# B&R Automation Studio project PLC_base3
Automation Studio 4.8.2.72

## Logical view

### Global.var - Global variables
```iecst
VAR
	data1 : STRING[1000];
	data2 : STRING[1000];
	activeData : USINT;
	readyForData : BOOL;
	receivedData : BOOL;
	readyToConvert : BOOL;
	instSize : DINT;
	instructionsArray : ARRAY[0..999] OF STRING[25];
	xArray : ARRAY[0..999] OF INT;
	yArray : ARRAY[0..999] OF INT;
	zArray : ARRAY[0..999] OF INT;
END_VAR
```

### Program Logical/Program (IEC)

#### Main.st - Init, cyclic, exit code
```iecst
PROGRAM _INIT
	ROBOSTATE := READY;

	counter := 0;
	delim1 := ' ';
	delim2 := ',';

	xEnable := FALSE;
	yEnable := FALSE;
	zEnable := FALSE;

	count := 0;
	xCounter := 0;
	yCounter := 0;
	zCounter := 0;
	xCalib := 0; //17680
	yCalib := 0; //13364
	zCalib := 0;
	yPrev := 0;
	xNext := FALSE;
	yNext := FALSE;
	zNext := FALSE;
	xDirection := FALSE;
	yDirection := FALSE;
	zDirection := FALSE;
	xStep := FALSE;
	yStep := FALSE;
	zStep := FALSE;
	xNegMove := FALSE;
	yNegMove := FALSE;
	zNegMove := FALSE;
	xPosMove := FALSE;
	yPosMove := FALSE;
	zPosMove := FALSE;
	hasBeenSharpened := TRUE;
	scale := 25; // steps / px
END_PROGRAM

PROGRAM _CYCLIC
	IF killswitch THEN // Killswitch to stop robot in case of emergency
		//ROBOSTATE := STOP;
	END_IF;

	CASE ROBOSTATE OF
		INIT:
			counter := 0;
			delim1 := ' ';
			delim2 := ',';

			xEnable := FALSE;
			yEnable := FALSE;
			zEnable := FALSE;

			count := 0;
			xCounter := 0;
			yCounter := 0;
			zCounter := 0;
			xCalib := 0; //17680
			yCalib := 0; //13364
			zCalib := 0;
			yPrev := 0;
			xNext := FALSE;
			yNext := FALSE;
			zNext := FALSE;
			xDirection := FALSE;
			yDirection := FALSE;
			zDirection := FALSE;
			xStep := FALSE;
			yStep := FALSE;
			zStep := FALSE;
			xNegMove := FALSE;
			yNegMove := FALSE;
			zNegMove := FALSE;
			xPosMove := FALSE;
			yPosMove := FALSE;
			zPosMove := FALSE;
			readyToConvert := FALSE;
			scale := 25;

			FOR count := 0 TO 999 DO
				instructionsArray[count] := '';
				xArray[count] := 0;
				yArray[count] := 0;
				zArray[count] := 0;
			END_FOR;

			ROBOSTATE := READY;

		READY: // Does nothing, is meant to wait until finished receiving instructions
			IF (readyToConvert = TRUE) THEN
				ROBOSTATE := CONVERT;
			END_IF

		CONVERT:
			timer(IN := NOT timer.Q, PT := T#100ms);
			IF (timer.Q = TRUE) THEN
				IF (counter < (instSize)) THEN
					// Splits element on index counter of instructionsArray[] into two seperate strings
					string1 := LEFT(instructionsArray[counter], FIND(instructionsArray[counter], delim2));
					string2 := RIGHT(instructionsArray[counter], (LEN(instructionsArray[counter]) - FIND(instructionsArray[counter], delim2)));

					// Finds numerical positions of all delimiters " " and "," in both strings
					// Isolates coordinates into individual integers
					D1 := FIND(string1, delim1);
					xString[counter] := LEFT(string1, D1 - 1);
					xArray[counter] := STRING_TO_INT(xString[counter]);
					string1 := DELETE(string1, D1, 1);

					D2 := FIND(string1, delim1);
					yString[counter] := LEFT(string1, D2 - 1);
					yArray[counter] := STRING_TO_INT(yString[counter]);
					string1 := DELETE(string1, D2, 1);

					D3 := FIND(string1, delim2);
					zString[counter] := LEFT(string1, D3 - 1);
					zArray[counter] := STRING_TO_INT(zString[counter]);

					D4 := FIND(string2, delim1);
					xString[counter + 1] := LEFT(string2, D4 - 1);
					xArray[counter + 1] := STRING_TO_INT(xString[counter + 1]);
					string2 := DELETE(string2, D1, 1);

					D5 := FIND(string2, delim1);
					yString[counter + 1] := LEFT(string2, D5 - 1);
					yArray[counter + 1] := STRING_TO_INT(yString[counter + 1]);
					string2 := DELETE(string2, D2, 1);

					D6 := FIND(string2, delim2);
					zString[counter + 1] := LEFT(string2, D6 - 1);
					zArray[counter + 1] := STRING_TO_INT(zString[counter + 1]);
					counter := counter + 2;
				ELSE
					ROBOSTATE := RESET;

					counter := 0;
				END_IF
			END_IF

		MANUAL:
			IF (killswitch <> TRUE) THEN
				IF (xStop <> TRUE OR xCounter > 0) THEN
					IF (xPosMove = TRUE) THEN
						IF (xPosMove = xNegMove) THEN
							xPosMove := FALSE;
						END_IF
						xDirection := TRUE;
						xStep := NOT xStep;
						xCounter := xCounter + 1;
					END_IF

					IF (xNegMove = TRUE) THEN
						IF (xPosMove = xNegMove) THEN
							xNegMove := FALSE;
						END_IF
						xDirection := FALSE;
						xStep := NOT xStep;
						xCounter := xCounter - 1;
					END_IF
				END_IF

				IF (yStop <> TRUE OR yCounter > 0) THEN
					IF (yPosMove = TRUE) THEN
						IF (yPosMove = yNegMove) THEN
							yPosMove := FALSE;
						END_IF
						yDirection := TRUE;
						yStep := NOT yStep;
						yCounter := yCounter + 1;
					END_IF

					IF (yNegMove = TRUE) THEN
						IF (yPosMove = yNegMove) THEN
							yNegMove := FALSE;
						END_IF
						yDirection := FALSE;
						yStep := NOT yStep;
						yCounter := yCounter - 1;
					END_IF
				END_IF

				IF (zCounter >= 0 AND zCounter <= 7500) THEN
					IF (zPosMove = TRUE) THEN
						IF (zPosMove = zNegMove) THEN
							zPosMove := FALSE;
						END_IF
						zDirection := TRUE;
						zStep := NOT zStep;
						zCounter := zCounter - 1;
					END_IF

					IF (zNegMove = TRUE) THEN
						IF (zPosMove = zNegMove) THEN
							zNegMove := FALSE;
						END_IF
						zDirection := FALSE;
						zStep := NOT zStep;
						zCounter := zCounter + 1;
					END_IF
				END_IF
			END_IF

		DRAW:
			IF (killswitch <> TRUE) OR (counter < instSize) THEN
				IF (xStop <> TRUE) THEN
					IF (xArray[counter] * scale > xCounter) THEN
						xNext := FALSE;
						xDirection := TRUE;
						xStep := NOT xStep;
						xCounter := xCounter + 1;
					ELSIF (xArray[counter] * scale < xCounter) THEN
						xNext := FALSE;
						xDirection := FALSE;
						xStep := NOT xStep;
						xCounter := xCounter - 1;
					ELSIF (xArray[counter] * scale = xCounter) THEN
						ROBOSTATE := PENCILDOWN;
					END_IF
				END_IF
			END_IF

		PENCILDOWN:
			IF (killswitch <> TRUE) THEN
				IF (bStop <> TRUE) THEN
					zDirection := TRUE;
					zStep := NOT zStep;
					zCounter := zCounter - 1;
				ELSE
					ROBOSTATE := DRAW2;
				END_IF
			END_IF

		DRAW2:
			IF (killswitch <> TRUE) THEN
				IF (xStop <> TRUE) THEN
					IF (xArray[counter + 1] * scale > xCounter) THEN
						xDirection := TRUE;
						xStep := NOT xStep;
						xCounter := xCounter + 1;
					ELSIF (xArray[counter + 1] * scale < xCounter) THEN
						xDirection := FALSE;
						xStep := NOT xStep;
						xCounter := xCounter - 1;
					ELSIF (xArray[counter + 1] * scale = xCounter) THEN
						ROBOSTATE := PENCILUP;
					END_IF
				END_IF
			END_IF

		PENCILUP:
			IF (killswitch <> TRUE) THEN
				IF (zCounter < 500) THEN
					zDirection := FALSE;
					zStep := NOT zStep;
					zCounter := zCounter + 1;
				ELSIF (zCounter = 500) THEN
					counter := counter + 1;
					ROBOSTATE := NEXTLINE;
				END_IF
			END_IF

		CHECKLINE:
			IF (killswitch <> TRUE) THEN
				IF (yArray[counter + 1] = yArray[counter]) THEN
					ROBOSTATE := DRAW;
				ELSIF (yArray[counter + 1] <> yArray[counter]) THEN
					ROBOSTATE := NEXTLINE;
				END_IF
			END_IF

		NEXTLINE:
			IF (killswitch <> TRUE) THEN
				IF (yStop <> TRUE) THEN
					IF (yCounter = ((counter + 1) * scale)) THEN
						IF (hasBeenSharpened = FALSE) AND (counter MOD(50) = 0) THEN
							ROBOSTATE := SHARPEN;
						ELSE
							ROBOSTATE := DRAW;
						END_IF
					ELSIF (yCounter < ((counter + 1) * scale)) THEN
						yDirection := TRUE;
						yStep := NOT yStep;
						yCounter := yCounter + 1;
					END_IF
				END_IF
			END_IF

		SHARPEN:
			IF (killswitch <> TRUE) THEN
				IF (zCounter < 3500 AND zStop <> TRUE AND xStop <> TRUE) THEN
					zDirection := FALSE;
					zStep := NOT zStep;
					zCounter := zCounter + 1;
				ELSIF (zCounter >= 3500 AND xStop <> TRUE AND zStop <> TRUE) THEN
					xDirection := FALSE;
					xStep := NOT xStep;
					xCounter := xCounter - 1;
				ELSIF (xStop = TRUE AND zStop <> TRUE) THEN
					IF (hasBeenSharpened <> TRUE AND zCounter > 1450) THEN
						sharpener := TRUE;
						zDirection := TRUE;
						zStep := NOT zStep;
						zCounter := zCounter - 1;
					ELSIF (zCounter = 1450) THEN
						timer(IN := NOT timer.Q, PT := T#2500ms);
						hasBeenSharpened := TRUE;
					END_IF
					IF (zCounter < 3500 AND hasBeenSharpened = TRUE AND timer.Q) THEN
						sharpener := FALSE;
						zDirection := FALSE;
						zStep := NOT zStep;
						zCounter := zCounter + 1;
					ELSIF (zCounter >= 3500 AND hasBeenSharpened = TRUE) THEN
						ROBOSTATE := BACK;
					END_IF
				END_IF
			END_IF

		BACK:
			IF (killswitch <> TRUE) THEN
				IF (xArray[counter] * scale > xCounter AND hasBeenSharpened = TRUE) THEN
					xDirection := TRUE;
					xStep := NOT xStep;
					xCounter := xCounter + 1;
				ELSIF (xArray[counter] * scale = xCounter AND bStop <> TRUE AND hasBeenSharpened = TRUE) THEN
					zDirection := TRUE;
					zStep := NOT zStep;
					zCounter := zCounter - 1;
				ELSIF (xArray[counter] * scale = xCounter AND bStop = TRUE AND hasBeenSharpened = TRUE) THEN
					ROBOSTATE := DRAW;
				END_IF
			END_IF

		RESET: // ASSUMES XCALIB AND YCALIB AS CONTAINING MAX STEPS ON X AND Y AXIS AS IT USES THESE TO FIND ORIGO
			sharpener := FALSE;
			IF (killswitch <> TRUE) THEN
				zCalib := 0;
				IF (zStop <> TRUE) THEN
					zDirection := FALSE;
					zStep := NOT zStep;
					zCounter := zCounter + 1;
				ELSE
					zCounter := zCalib;
				END_IF
				IF (xStop <> TRUE AND zStop = TRUE) THEN
					xDirection := FALSE;
					xStep := NOT xStep;
					xCounter := xCounter + 1;
				ELSE
					xCounter := xCalib;
				END_IF
				IF (yStop <> TRUE AND zStop = TRUE) THEN
					yDirection := FALSE;
					yStep := NOT yStep;
					yCounter := yCounter + 1;
				ELSE
					yCounter := yCalib;
				END_IF

				IF (xStop = TRUE AND yStop = TRUE AND zStop = TRUE) THEN
					ROBOSTATE := CALIBRATE;
				END_IF
			END_IF

		CALIBRATE: // ONLY USE CALIBRATE IF ALL STOP SENSORS ARE ACTIVATED
			IF (xCounter < 3280) THEN
				xDirection := TRUE;
				xStep := NOT xStep;
				xCounter := xCounter + 1;
			END_IF
			IF (yCounter < 1364) THEN
				yDirection := TRUE;
				yStep := NOT yStep;
				yCounter := yCounter + 1;
			END_IF
			IF (xCounter >= 3280 AND xCounter <= 17680 AND yCounter >= 1364 AND yCounter <= 13364) THEN
				IF (bStop <> TRUE AND zPosMove = FALSE) THEN
					zDirection := TRUE;
					zStep := NOT zStep;
					zCounter := zCounter + 1;
				ELSIF (bStop = TRUE AND zPosMove = FALSE) THEN
					zPosMove := TRUE;
					zCounter := 0;
				ELSIF (zPosMove = TRUE) THEN
					IF (zCounter < 500) THEN
						zDirection := FALSE;
						zStep := NOT zStep;
						zCounter := zCounter + 1;
					ELSE
						zPosMove := FALSE;
						xCounter := 0;
						yCounter := 0;
						ROBOSTATE := MANUAL;
					END_IF
				END_IF
			END_IF
	END_CASE
END_PROGRAM

PROGRAM _EXIT

END_PROGRAM
```

#### COORD_TO_STEP.st
```iecst
(* Omdanner et koordinat til et antal steps *)
FUNCTION COORD_TO_STEP
	STEP_COUNT := COORD * 25;
END_FUNCTION
```

### Program Logical/Socket (IEC)

#### Types.typ
```iecst
TYPE
	RESETSTATE :
		(
		RUN,
		RESET
		);
	TCPSTATE :
		(
		TCPSTATE_CLOSE,
		TCPSTATE_SEND,
		TCPSTATE_RECEIVE,
		TCPSTATE_SERVER_CREATE,
		TCPSTATE_SOCKET_OPEN,
		TCPSTATE_RESET
		);
END_TYPE
```

Listed in the project but not available here: Logical/Global.typ, Logical/Program/Types.typ, Logical/Program/Variables.var, Logical/Program/LocalFunctions.fun
